FUNCTION_BLOCK M_SET (* Matrix Setup *)
  (* Standard: 61499-1; Classification: Matrix Operations; Function: Initialization *)
  (* Version 0.0, 2002-03-07, JHC, Rockwell Automation *)
  (* Compiler header: package fb.rt.math; *)
  (* Compiler Java IBM VisualAge 3.0 *)
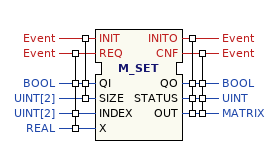
  EVENT_INPUT
    INIT WITH QI, SIZE; (* Set OUT to zeroes of extent SIZE *)
    REQ WITH QI, INDEX, X; (* Replace data at INDEX by value of X *)
  END_EVENT
  EVENT_OUTPUT
    INITO WITH QO, STATUS, OUT;
    CNF WITH QO, STATUS, OUT;
  END_EVENT
  VAR_INPUT
    QI : BOOL; (* 0=Inhibit,1=Enable *)
    SIZE : ARRAY [0..1] OF UINT; (* Number of[rows,columns] *)
    INDEX : ARRAY [0..1] OF UINT; (* [row,column] *)
    X : REAL; (* Data for INDEX location *)
  END_VAR
  VAR_OUTPUT
    QO : BOOL; (* 1=OK,0=Inhibited or Error *)
    STATUS : UINT; (* 0=OK,1=INHIBITED,13=ARRAY_SIZE_ERROR *)
    OUT : MATRIX;
  END_VAR
END_FUNCTION_BLOCK
